FUNCTION_BLOCK FB_Sequence IMPLEMENTS I_Sequence
VAR_INPUT
	bHeld:				BOOL;
END_VAR
VAR_OUTPUT
	bTimeout:			BOOL;
END_VAR
VAR
	iParent:			I_Element;
	stExecute:			ST_Sequence;
	stLast:				ST_Sequence;
	stActual:			ST_Sequence;
	fbTimeout:			TON;
	fbDelay: 			TON;
END_VAR

// https://peterzerlauth.com/

METHOD FB_init : BOOL
VAR_INPUT
	bInitRetains : BOOL; // if TRUE, the retain variables are initialized (warm start / cold start)
	bInCopyCode : BOOL;  // if TRUE, the instance afterwards gets moved into the copy code (online change)
	iParent:			I_Element;
END_VAR
THIS^.iParent:= iParent;
END_METHOD

METHOD PUBLIC M_Await : BOOL
VAR_INPUT
	sMessage:				STRING(255);
	nID:					ULINT;
	tTimeout:				TIME;
	tDelay:					TIME;	
	bPause:					BOOL;
	bReturn:				BOOL;
	nNumber:				INT;
END_VAR
// Assign the current message to the actual status structure
stActual.sMessage := sMessage;  

// Check the return condition
IF bReturn THEN  
    // Reset timeout
    fbTimeout(IN := FALSE);  
    bTimeout := FALSE; 
    // Start delay
    fbDelay(IN := TRUE, PT := tDelay);  
    
    // Delay elapsed  
    IF fbDelay.Q THEN  
        M_Await := TRUE;  
        // Set the next step number
        stActual.nNumber := nNumber;   
        // Save the last known state  
        stLast := stActual;  
        // Last state to restore
        IF iParent.P_State = E_State.Execute THEN  
            stExecute := stLast;  
        END_IF  
        
        // Reset delay
        fbDelay(IN := FALSE);  
//         IF bHeld THEN  
//             // Request a hold operation to the parent  
//             iParent.M_Request(E_Request.Hold);  
//         ELSIF bPause THEN  
//             // Request a pause operation to the parent  
//             iParent.M_Request(E_Request.Pause);  
//         END_IF  
    END_IF  

ELSE  
    // Reset delay
    fbDelay(IN := FALSE);  
    // Start timeout
    fbTimeout(IN := tTimeout <> T#0S, PT := tTimeout);  
    // Timeout elapsed
    IF fbTimeout.Q THEN
		bTimeout := TRUE;   
        // Report Timeout 
        iParent.P_Event.M_Error(sMessage, nID);  
    END_IF  
END_IF
END_METHOD

METHOD PUBLIC M_Reset : BOOL
VAR_INPUT
END_VAR
bTimeout:= FALSE;
fbDelay(IN:= FALSE);
fbTimeout(IN:= FALSE);
stActual.sMessage:= 'fbSequence.M_Reset()';
stActual.nNumber:= E_Sequence.Start;
M_Reset:= TRUE;
END_METHOD

METHOD PUBLIC M_Restore : BOOL
VAR_INPUT
END_VAR
stLast:= stActual;
stActual:= stExecute;
END_METHOD

METHOD PUBLIC M_Set : BOOL
VAR_INPUT
	sMessage:				STRING(255);	
	nNumber:				INT;
END_VAR
stLast:= stActual;
IF iParent.P_State = E_State.Execute THEN
	stExecute:= stActual;
END_IF
stActual.sMessage:= Concat('Sequence.M_Set: ', sMessage);
stActual.nNumber:= nNumber;
M_Set:= TRUE;
END_METHOD


PROPERTY PUBLIC P_Number : INT
GET
P_Number:= stActual.nNumber;
END_GET
END_PROPERTY

PROPERTY PUBLIC P_Timeout : Bool
GET
P_Timeout:= bTimeout;
END_GET
END_PROPERTY

END_FUNCTION_BLOCK

(* stored: Version 1.1.0.1
   POU FB_Sequence: Id {4b1aa270-5e63-4fbf-b9b1-b64186ed4cc4}, SpecialFunc None
   Method FB_init: Id {9410888f-1e8d-054b-01cb-f8f70c408f51}
   Method M_Await: Id {1bc0e82b-8467-4f35-a54e-996600fba2bc}
   Method M_Reset: Id {36513383-9494-0732-02c6-f9c957e037d9}
   Method M_Restore: Id {1bd7bf81-b107-0061-0190-e2f9ae962872}
   Method M_Set: Id {1679b774-aff9-0900-1b9f-6b982123f170}
   Property P_Number: Id {3cc751bf-6092-4aa8-8de5-3276200b64ad}
   Get Get: Id {92b3a1f5-52d3-44fe-8629-e1295a1ef489}
   Property P_Timeout: Id {eb074bec-3376-04de-22f4-48dc23a1d0c0}
   Get Get: Id {4091acc7-d1a3-074a-2f14-85ba09be9e4b} *)
